FUNCTION_BLOCK FB_DataToNovRam
VAR_INPUT
	bExecute:BOOL;
	
	savedData:ST_AlarmInfo_DB_save;
END_VAR
VAR_OUTPUT
	bResult:BOOL;
END_VAR
VAR
	
END_VAR
VAR_IN_OUT
END_VAR

METHOD M_AlarmHistory : BOOL
VAR_INPUT
	addData:ST_AlarmInfo_DB;
END_VAR
VAR
	eStrIndex:DINT;
	udiNowRowIndex:DINT;
	udiWritenIndex:DINT;
	CompressedData:ST_AlarmInfo_DB_save;
END_VAR
//Config
eStrIndex:=E_StructureType.AlarmHistory;
udiNowRowIndex:=GVL.NovRamData.arrNovRam_Status[eStrIndex].nowRowIndex;
udiWritenIndex:=GVL.NovRamData.arrNovRam_Status[eStrIndex].writenIndex;

IF GVL.NovRamData.arrNovRam_Status[eStrIndex].RowDataLocked[udiNowRowIndex]=FALSE THEN//writable
	
	//write data
	M_ST_AlarmHistory_Compress(Input:=addData,Output=>GVL.NovRamData.AlarmHistory[udiNowRowIndex][udiWritenIndex]);
	
	GVL.NovRamData.arrNovRam_Status[eStrIndex].writenIndex:=GVL.NovRamData.arrNovRam_Status[eStrIndex].writenIndex+1;
	
	//Check if Full
	IF GVL.NovRamData.arrNovRam_Status[eStrIndex].writenIndex >= (GVL.arrArrayLength[eStrIndex] - 1) THEN
		//Set Row Lock
		GVL.NovRamData.arrNovRam_Status[eStrIndex].RowDataLocked[udiNowRowIndex]:=TRUE;
		
		//Reset Row and writenIndex
		GVL.NovRamData.arrNovRam_Status[eStrIndex].nowRowIndex:=(udiNowRowIndex+1)MOD GVL.NovRamBufferRatio;
		GVL.NovRamData.arrNovRam_Status[eStrIndex].writenIndex:=0;
	END_IF
	
	M_AlarmHistory:=TRUE;
ELSE
	M_AlarmHistory:=FALSE;
END_IF
END_METHOD

METHOD M_ProductionHistory : BOOL
VAR_INPUT
	addData:ST_PHI_GroupData_DB;
END_VAR
VAR 
	eStrIndex:DINT;
	udiNowRowIndex:DINT;
	udiWritenIndex:DINT;
	CompressedData:ST_PHI_GroupData_DB;
END_VAR
//Config
eStrIndex:=E_StructureType.ProductionHistory;
udiNowRowIndex:=GVL.NovRamData.arrNovRam_Status[eStrIndex].nowRowIndex;
udiWritenIndex:=GVL.NovRamData.arrNovRam_Status[eStrIndex].writenIndex;

IF GVL.NovRamData.arrNovRam_Status[eStrIndex].RowDataLocked[udiNowRowIndex]=FALSE THEN//writable
	
	//write data
	M_ST_ProductionHistory_Compress(Input:=addData,Output=>GVL.NovRamData.ProductionHistory[udiNowRowIndex][udiWritenIndex]);
	
	GVL.NovRamData.arrNovRam_Status[eStrIndex].writenIndex:=GVL.NovRamData.arrNovRam_Status[eStrIndex].writenIndex+1;
	
	//Check if Full
	IF GVL.NovRamData.arrNovRam_Status[eStrIndex].writenIndex >= (GVL.arrArrayLength[eStrIndex] - 1) THEN
		//Set Row Lock
		GVL.NovRamData.arrNovRam_Status[eStrIndex].RowDataLocked[udiNowRowIndex]:=TRUE;
		
		//Reset Row and writenIndex
		GVL.NovRamData.arrNovRam_Status[eStrIndex].nowRowIndex:=(udiNowRowIndex+1)MOD GVL.NovRamBufferRatio;
		GVL.NovRamData.arrNovRam_Status[eStrIndex].writenIndex:=0;
	END_IF
	
	M_ProductionHistory:=TRUE;
ELSE
	M_ProductionHistory:=FALSE;
END_IF
END_METHOD

METHOD M_ProductionReport : BOOL
VAR_INPUT
	addData:ST_OEE_ProductionReport;
END_VAR
VAR
	eStrIndex:DINT;
	udiNowRowIndex:DINT;
	udiWritenIndex:DINT;
	CompressedData:ST_OEE_ProductionReport;
END_VAR
//Config
eStrIndex:=E_StructureType.ProductionReport;
udiNowRowIndex:=GVL.NovRamData.arrNovRam_Status[eStrIndex].nowRowIndex;
udiWritenIndex:=GVL.NovRamData.arrNovRam_Status[eStrIndex].writenIndex;

IF GVL.NovRamData.arrNovRam_Status[eStrIndex].RowDataLocked[udiNowRowIndex]=FALSE THEN//writable
	
	//write data
	M_ST_ProductionReport_Compress(Input:=addData,Output=>GVL.NovRamData.ProductionReport[udiNowRowIndex][udiWritenIndex]);

	GVL.NovRamData.arrNovRam_Status[eStrIndex].writenIndex:=GVL.NovRamData.arrNovRam_Status[eStrIndex].writenIndex+1;
	
	//Check if Full
	IF GVL.NovRamData.arrNovRam_Status[eStrIndex].writenIndex >= (GVL.arrArrayLength[eStrIndex] - 1) THEN
		//Set Row Lock
		GVL.NovRamData.arrNovRam_Status[eStrIndex].RowDataLocked[udiNowRowIndex]:=TRUE;
		
		//Reset Row and writenIndex
		GVL.NovRamData.arrNovRam_Status[eStrIndex].nowRowIndex:=(udiNowRowIndex+1)MOD GVL.NovRamBufferRatio;
		GVL.NovRamData.arrNovRam_Status[eStrIndex].writenIndex:=0;
	END_IF
	
	M_ProductionReport:=TRUE;
ELSE
	M_ProductionReport:=FALSE;
END_IF
END_METHOD

METHOD M_ProductionSummary : BOOL
VAR_INPUT
	addData:ST_OEE_ProductionSummary;
END_VAR
VAR
	eStrIndex:DINT;
	udiNowRowIndex:DINT;
	udiWritenIndex:DINT;
	CompressedData:ST_OEE_ProductionSummary;
END_VAR
//Config
eStrIndex:=E_StructureType.ProductionSummary;
udiNowRowIndex:=GVL.NovRamData.arrNovRam_Status[eStrIndex].nowRowIndex;
udiWritenIndex:=GVL.NovRamData.arrNovRam_Status[eStrIndex].writenIndex;

IF GVL.NovRamData.arrNovRam_Status[eStrIndex].RowDataLocked[udiNowRowIndex]=FALSE THEN//writable
	
	//write data
	M_ST_ProductionSummary_Compress(Input:=addData,Output=>GVL.NovRamData.ProductionSummary[udiNowRowIndex][udiWritenIndex]);

	GVL.NovRamData.arrNovRam_Status[eStrIndex].writenIndex:=GVL.NovRamData.arrNovRam_Status[eStrIndex].writenIndex+1;
	
	//Check if Full
	IF GVL.NovRamData.arrNovRam_Status[eStrIndex].writenIndex >= (GVL.arrArrayLength[eStrIndex] - 1) THEN
		//Set Row Lock
		GVL.NovRamData.arrNovRam_Status[eStrIndex].RowDataLocked[udiNowRowIndex]:=TRUE;
		
		//Reset Row and writenIndex
		GVL.NovRamData.arrNovRam_Status[eStrIndex].nowRowIndex:=(udiNowRowIndex+1)MOD GVL.NovRamBufferRatio;
		GVL.NovRamData.arrNovRam_Status[eStrIndex].writenIndex:=0;
	END_IF
	
	M_ProductionSummary:=TRUE;
ELSE
	M_ProductionSummary:=FALSE;
END_IF
END_METHOD

METHOD M_RegularCheckResults : BOOL
VAR_INPUT
	addData:ST_RegularCheck_Results;
END_VAR
VAR
	eStrIndex:DINT;
	udiNowRowIndex:DINT;
	udiWritenIndex:DINT;
	CompressedData:ST_RegularCheck_Results;
END_VAR
//Config
eStrIndex:=E_StructureType.RegularCheckResults;
udiNowRowIndex:=GVL.NovRamData.arrNovRam_Status[eStrIndex].nowRowIndex;
udiWritenIndex:=GVL.NovRamData.arrNovRam_Status[eStrIndex].writenIndex;

IF GVL.NovRamData.arrNovRam_Status[eStrIndex].RowDataLocked[udiNowRowIndex]=FALSE THEN//writable
	
	//write data
	M_ST_RegularCheckResults_Compress(Input:=addData,Output=>GVL.NovRamData.RegularCheckResults[udiNowRowIndex][udiWritenIndex]);
	
	GVL.NovRamData.arrNovRam_Status[eStrIndex].writenIndex:=GVL.NovRamData.arrNovRam_Status[eStrIndex].writenIndex+1;
	
	//Check if Full
	IF GVL.NovRamData.arrNovRam_Status[eStrIndex].writenIndex >= (GVL.arrArrayLength[eStrIndex] - 1) THEN
		//Set Row Lock
		GVL.NovRamData.arrNovRam_Status[eStrIndex].RowDataLocked[udiNowRowIndex]:=TRUE;
		
		//Reset Row and writenIndex
		GVL.NovRamData.arrNovRam_Status[eStrIndex].nowRowIndex:=(udiNowRowIndex+1)MOD GVL.NovRamBufferRatio;
		GVL.NovRamData.arrNovRam_Status[eStrIndex].writenIndex:=0;
	END_IF
	
	M_RegularCheckResults:=TRUE;
ELSE
	M_RegularCheckResults:=FALSE;
END_IF
END_METHOD

METHOD M_SoDuration : BOOL
VAR_INPUT
	addData:ST_SoDuration;
END_VAR
VAR
	eStrIndex:DINT;
	udiNowRowIndex:DINT;
	udiWritenIndex:DINT;
	CompressedData:ST_SoDuration;
END_VAR
//Config
eStrIndex:=E_StructureType.SoDuration;
udiNowRowIndex:=GVL.NovRamData.arrNovRam_Status[eStrIndex].nowRowIndex;
udiWritenIndex:=GVL.NovRamData.arrNovRam_Status[eStrIndex].writenIndex;

IF GVL.NovRamData.arrNovRam_Status[eStrIndex].RowDataLocked[udiNowRowIndex]=FALSE THEN//writable
	
	//write data
	M_ST_SoDuration_Compress(Input:=addData,Output=>GVL.NovRamData.SoDuration[udiNowRowIndex][udiWritenIndex]);
	
	GVL.NovRamData.arrNovRam_Status[eStrIndex].writenIndex:=GVL.NovRamData.arrNovRam_Status[eStrIndex].writenIndex+1;
	
	//Check if Full
	IF GVL.NovRamData.arrNovRam_Status[eStrIndex].writenIndex >= (GVL.arrArrayLength[eStrIndex] - 1) THEN
		//Set Row Lock
		GVL.NovRamData.arrNovRam_Status[eStrIndex].RowDataLocked[udiNowRowIndex]:=TRUE;
		
		//Reset Row and writenIndex
		GVL.NovRamData.arrNovRam_Status[eStrIndex].nowRowIndex:=(udiNowRowIndex+1)MOD GVL.NovRamBufferRatio;
		GVL.NovRamData.arrNovRam_Status[eStrIndex].writenIndex:=0;
	END_IF
	
	M_SoDuration:=TRUE;
ELSE
	M_SoDuration:=FALSE;
END_IF
END_METHOD

METHOD M_ST_AlarmHistory_Compress : BOOL
VAR_INPUT
	Input:ST_AlarmInfo_DB;
END_VAR
VAR_OUTPUT
	Output:ST_AlarmInfo_DB_save;
END_VAR
Output.lrTime_ms:=Input.lrTime_ms;
Output.iMsgProc:=Input.iMsgProc;
Output.iStateAfter:=Input.iStateAfter;
Output.iMsgClass:=Input.iMsgClass;
Output.diMsgNumber:=Input.diMsgNumber;
Output.sTimeString:=Input.sTimeString;
Output.wsMsgText:=Input.wsMsgText;
Output.sPLC:=Input.sPLC;
Output.wsEquipment:=Input.wsEquipment;
Output.sFaam_id:=Input.sFaam_id;
END_METHOD

METHOD M_ST_ProductionHistory_Compress : BOOL
VAR_INPUT
	Input:ST_PHI_GroupData_DB;
END_VAR
VAR_OUTPUT
	Output:ST_PHI_GroupData_DB;
END_VAR
Output:=Input;
END_METHOD

METHOD M_ST_ProductionReport_Compress : BOOL
VAR_INPUT
	Input:ST_OEE_ProductionReport;
END_VAR
VAR_OUTPUT
	Output:ST_OEE_ProductionReport;
END_VAR
Output:=Input;
END_METHOD

METHOD M_ST_ProductionSummary_Compress : BOOL
VAR_INPUT
	Input:ST_OEE_ProductionSummary;
END_VAR
VAR_OUTPUT
	Output:ST_OEE_ProductionSummary;
END_VAR
Output:=Input;
END_METHOD

METHOD M_ST_RegularCheckResults_Compress : BOOL
VAR_INPUT
	Input:ST_RegularCheck_Results;
END_VAR
VAR_OUTPUT
	Output:ST_RegularCheck_Results;
END_VAR
(*
Output.stProductHistory.diStation_number:=Input.stProductHistory.diStation_number;
Output.stProductHistory.diTrack_number:=Input.stProductHistory.diTrack_number;
Output.stProductHistory.dtStart_time:=Input.stProductHistory.dtStart_time;

IF Input.bSensor = TRUE THEN
	Output.eSensor:=E_RegularCheckSensorResult.Pass;
ELSE
	Output.eSensor:=E_RegularCheckSensorResult.Fail;
END_IF

IF Input.bCamera = TRUE THEN
	Output.eCamera:=E_RegularCheckSensorResult.Pass;
ELSE
	Output.eCamera:=E_RegularCheckSensorResult.Fail;
END_IF

IF Input.bLoadcell = TRUE THEN
	Output.eLoadcell:=E_RegularCheckSensorResult.Pass;
ELSE
	Output.eLoadcell:=E_RegularCheckSensorResult.Fail;
END_IF

IF Input.bSensor2 = TRUE THEN
	Output.eSensor2:=E_RegularCheckSensorResult.Pass;
ELSE
	Output.eSensor2:=E_RegularCheckSensorResult.Fail;
END_IF

Output.diRegular_check_id:=Input.diRegular_check_id;
Output.sFaam_id:=Input.sFaam_id;
Output.sSo_number:=Input.sSo_number;
Output.diSo_id:=Input.diSo_id;
Output.wsEmployee_name_logged_in:=Input.wsEmployee_name_logged_in;
*)
Output:=Input;
END_METHOD

METHOD M_ST_SoDuration_Compress : BOOL
VAR_INPUT
	Input:ST_SoDuration;
END_VAR
VAR_OUTPUT
	Output:ST_SoDuration;
END_VAR
Output:=Input;
END_METHOD

METHOD M_ST_StopCount_Compress : BOOL
VAR_INPUT
	Input:ST_StopCount;
END_VAR
VAR_OUTPUT
	Output:ST_StopCount;
END_VAR
Output:=Input;
END_METHOD

METHOD M_StopCount : BOOL
VAR_INPUT
	addData:ST_StopCount;
END_VAR
VAR
	eStrIndex:DINT;
	udiNowRowIndex:DINT;
	udiWritenIndex:DINT;
	CompressedData:ST_StopCount;
END_VAR
//Config
eStrIndex:=E_StructureType.StopCount;
udiNowRowIndex:=GVL.NovRamData.arrNovRam_Status[eStrIndex].nowRowIndex;
udiWritenIndex:=GVL.NovRamData.arrNovRam_Status[eStrIndex].writenIndex;

IF GVL.NovRamData.arrNovRam_Status[eStrIndex].RowDataLocked[udiNowRowIndex]=FALSE THEN//writable
	
	//write data
	M_ST_StopCount_Compress(Input:=addData,Output=>GVL.NovRamData.StopCount[udiNowRowIndex][udiWritenIndex]);

	GVL.NovRamData.arrNovRam_Status[eStrIndex].writenIndex:=GVL.NovRamData.arrNovRam_Status[eStrIndex].writenIndex+1;
	
	//Check if Full
	IF GVL.NovRamData.arrNovRam_Status[eStrIndex].writenIndex >= (GVL.arrArrayLength[eStrIndex] - 1) THEN
		//Set Row Lock
		GVL.NovRamData.arrNovRam_Status[eStrIndex].RowDataLocked[udiNowRowIndex]:=TRUE;
		
		//Reset Row and writenIndex
		GVL.NovRamData.arrNovRam_Status[eStrIndex].nowRowIndex:=(udiNowRowIndex+1)MOD GVL.NovRamBufferRatio;
		GVL.NovRamData.arrNovRam_Status[eStrIndex].writenIndex:=0;
	END_IF
	
	M_StopCount:=TRUE;
ELSE
	M_StopCount:=FALSE;
END_IF
END_METHOD

END_FUNCTION_BLOCK

(* stored: Version 1.1.0.1, ProductVersion 3.1.4024.11
   POU FB_DataToNovRam: Id {76f3141b-7a21-4959-afa9-90d9594b687d}, SpecialFunc None
   Folder Sub: Id {2534213c-7e5e-4abf-9411-860d44a5b2d2}
   Method M_AlarmHistory: Id {aac47326-eba1-4863-89c8-9d8cb955d250}
   Method M_ProductionHistory: Id {d7343e0a-38fb-4763-8037-34bbcaf9758f}
   Method M_ProductionReport: Id {2687dc60-389f-4ef4-84c5-501218c7098f}
   Method M_ProductionSummary: Id {a4b2b19b-80fa-4785-b664-d0b380caa519}
   Method M_RegularCheckResults: Id {9aa594fd-a6f0-4775-b77b-92a3336da06a}
   Method M_SoDuration: Id {d9f5c0bb-6506-473d-93d1-a17c9d6d32f6}
   Method M_ST_AlarmHistory_Compress: Id {90234377-5e57-4a9c-9b48-a547d1d556f7}
   Method M_ST_ProductionHistory_Compress: Id {56b298ca-fed2-4f78-8add-9ff8f9eca520}
   Method M_ST_ProductionReport_Compress: Id {6448b315-2048-49f6-b778-7e67bf20eea8}
   Method M_ST_ProductionSummary_Compress: Id {8cecd652-1a50-4b26-88c4-1513f9101c97}
   Method M_ST_RegularCheckResults_Compress: Id {3d691fe0-8452-4cec-baed-830d96336e29}
   Method M_ST_SoDuration_Compress: Id {8efca6c8-584d-46e0-9bd4-7ed0f3c98d6e}
   Method M_ST_StopCount_Compress: Id {483d237d-5099-4da3-9f28-7308f5bcf526}
   Method M_StopCount: Id {60ce841c-0d92-4ca8-9d69-3454400f79f4} *)
